{attribute 'linkalways'} 
{attribute 'no_explicit_call' := 'This FB is a CLASS and must be accessed using methods or properties'}
{attribute 'enable_dynamic_creation'}
FUNCTION_BLOCK Node_ContainerType_String_SINT EXTENDS Node
VAR
    out : _GUID;
END_VAR

METHOD PUBLIC  Clone : I_Node
VAR
	pNode : POINTER TO Node_ContainerType_String_SINT;
END_VAR
pNode := __NEW(Node_ContainerType_String_SINT);
Clone := pNode^;
END_METHOD

METHOD FB_init : BOOL
VAR_INPUT
	bInitRetains : BOOL; // if TRUE, the retain variables are initialized (warm start / cold start)
	bInCopyCode : BOOL;  // if TRUE, the instance afterwards gets moved into the copy code (online change)
END_VAR
AddOutput('out', out);
END_METHOD

METHOD PROTECTED OnExecute
out.Value := ContainerType_String_SINT;
END_METHOD

END_FUNCTION_BLOCK

(* stored: Version 1.1.0.1, ProductVersion 3.1.4026.17
   POU Node_ContainerType_String_SINT: Id {9684099a-32fb-053b-3bcc-9f533b7ecbd3}, SpecialFunc None
   Folder Constructor: Id {b0bd7311-92ae-0b3e-0d74-09a8da5f191b}
   Method Clone: Id {c0ad2c5d-6f51-04f9-182e-f1572d849d18}
   Method FB_init: Id {1f6374ba-a9b3-0e33-1138-7f2be2159dca}
   Method OnExecute: Id {365a78a1-c71c-0431-223d-61797560770d} *)
